Staubli VAL3: ProductReady.pgx

public program ProductReady(num& x_nIndex (dimensions=1), bool x_bFirst (dimensions=1))
  local bool l_bRes
  local num l_nNum
  local string l_sStr
begin



  //2014.05.30
  //工位选择信号
  while true
    //第一工位
    for l_nNum=1 to 4
      if x_bFirst
        l_nNum=1
      endIf
      //测试
      if l_nNum==1 or l_nNum==2
        l_sStr="In1_bPrdSta"+toString("",l_nNum)
      endIf


      //第三工位或者第四工位用户可以进行自定义
      //××××××××××××××××××××××××××××××××××××××××
      if l_nNum==3
        l_sStr="In2_bPrdSta3"
      endIf

      if l_nNum==4
        l_sStr="In2_bPrdSta4"
      endIf
      //×××××××××××××××××××××××××××××××××××××××××
      //信号
      if dDio[l_sStr]==true
        delay(0.1)
        if watch(dDio[l_sStr]==true,0.1)
          logMsg("工位"+toString("",l_nNum)+"信号被触发")
          x_nIndex=l_nNum
          return
        endIf
      endIf

    endFor
    delay(0)
  endWhile



end
